Staubli VAL3: DataBase.dtx

public bool bAirOn
public bool bAlarm
public bool bDebugMode
public bool bExtraContrAxis
public bool bFollowOn
public bool bGasChoose
public bool bIOControl = true
public bool bIOStart
public bool bIsHome = true
public bool bKeyIO[3]
public bool bLaserOn
public bool bMoveTask
public bool bMultiNormal
public bool bMutexAxis
public bool bPowerOn = true
public bool bSaveTrajPoint
public bool bSingleAxisMode = true
public bool bStopPoll
public bool bStopSimul = true
public bool bThickPlatPunch
public bool bThickPlate
public bool bUpload
public bool bWaitFollowDone
public bool bWorldMove = true
public bool bWpFinishIOOut
public frame fFrame = {fatherId=world[0]}
public frame fJogContext = {fatherId=world[0]}
public frame fOffset = {fatherId=world[0]}
public jointRx jCurrentJoint = {j1=11.05, j2=30.63, j3=127.04, j4=11.92, j5=-68.09, j6=-3.11}
public mdesc mJHome = {tmax=166.666667, blend=off}
mdesc mNomSpeed
public num n1AxisOffset = 0.1
public num nActionID = 0.258567
public num nArrayCutAction[2]
public num nArrayX = 1
public num nArrayY = 1
public num nArrayZ = 1
public num nAsysAxisPer = 0.008
public num nAvgCutSpeed = 177.53368
public num nAxisOffset[2]
public num nCutLength = 393.307878
public num nCutTime = 3.117
public num nCycleCount
public num nCycleIndex
public num nCycleMode
public num nCycleTime = 36.639
public num nDebugData
public num nID
public num nInterfaceType = 7
public num nPartMove[3]
public num nPointType
public num nPollTime = 0.028
public num nPresetData[5]
  [1] = -100
public num nProductCount
public num nProductIndex
public num nRemoteProduct = 8888
public num nRobotSpeed
public num nSpeedPercent = 1
public num nTestData
public num nToolMode = 3
public num nTrajIndex = 1
public num nVersion = 3
public num nWeldActionId
public num nWeldEndOffset = 10
public num nWeldEndStart
public num nWeldEndTime = 9217.537
public num nWeldStartTime
public num nWorkPlaceButto = -1
public num nWorkPlaceCount
public num nWorkPlaceIndex
public num nWpMutiCount[10]
public num nWpProduct[5]
public pointRx pCurrentPoint = {x=1083.467345, y=182.728388, z=-429.922191, rx=0.992266, ry=-179.737388, rz=2.304169, shoulder=lefty, elbow=epositive, wrist=wnegative, fatherId=world[0]}
string sCustom
public string sProductName[10]
  [0] = "112222"
  [1] = "test20150408"
public string sSoftWareTime = "2015_02_03"
public string sVersion[8]
  [0] = "s7.9 - Dec 10 2015 - 10:53:01"
  [1] = "rx160l-S1"
  [2] = "floor"
  [3] = "?"
public trsf trOffset[3]
public trsf trTeachTemp = {z=300, rx=15}
